// TwinCAT 3 PLC project TwinCAT_OpenFramework_Timers
// Title: TwinCAT Open Framework Timers
// Company: Oleksandr Tiutyk FOP
// Author: Oleksandr Tiutyk
// ProjectVersion: 1.0.13.0
// Description: TwinCAT.OpenFramework object-oriented timer wrapper, works as task
// ProgramVersion: 3.1.4026.28
// libraries:
//   Tc2_Standard, * (Beckhoff Automation GmbH)
//   Tc2_System, * (Beckhoff Automation GmbH)
//   [TwinCAT Open Framework Core], * (Oleksandr Tiutyk FOP)
//   [TwinCAT Open Framework Tasks], * (Oleksandr Tiutyk FOP)
// project tree:
//   Internal/ CurrentNamespace.TcPOU, NamespaceExtractor.TcPOU
//   / ITimer.TcIO, Timer.TcPOU (not stored)
//   Version/ Global_Version.TcGVL
// (motion and I/O tree: see PLC project twincat_openframework_core)
// real-time tasks:
//   TASK PlcTask: cycle T#10ms, priority 20, ADS port 350
//   TASK TestTask: cycle T#10ms, priority 1, ADS port 351
//   TASK RunnerTestTask: cycle T#10ms, priority 2, ADS port 354
//   TASK HowToTask: cycle T#10ms, priority 22, ADS port 353
// variable links:

// ---- Version/Global_Version.TcGVL
{attribute 'TcGenerated'}
{attribute 'no-analysis'}
{attribute 'linkalways'}
// This function has been automatically generated from the project information.
VAR_GLOBAL CONSTANT
	{attribute 'const_non_replaced'}
	stLibVersion_TwinCAT_Open_Framework_Timers : ST_LibVersion := (iMajor := 1, iMinor := 0, iBuild := 13, iRevision := 0, nFlags := 0, sVersion := '1.0.13.0');
END_VAR

// ---- ITimer.TcIO
(*!
<summary>Exposes a task-driven timer's interval, observations and restart operation.</summary>
<description>
Drive the timer through the inherited task lifecycle. Reading observations does not advance time; the
implementation updates them while executing. Timer-specific TON behavior is documented by Timer.
</description>
*)
INTERFACE ITimer EXTENDS TOF_Tasks.ITask

{attribute 'monitoring' := 'call'}
(*!
<summary>Reports the timer's latest elapsed observation.</summary>
<description>
Reading does not update or consume the observation. For Timer this is TON.Q, retained after normal completion
until Reset or restart; it is not independently a successful task-completion result.
</description>
*)
PROPERTY Elapsed : BOOL
GET
END_GET
END_PROPERTY

{attribute 'monitoring' := 'call'}
(*!
<summary>Returns the latest elapsed-time observation without advancing the timer.</summary>
<description>
For Timer this is TON.ET from the most recent TON evaluation, not a live clock read. Reset clears the
observation.
</description>
*)
PROPERTY ElapsedTime : TIME
GET
END_GET
END_PROPERTY

{attribute 'monitoring' := 'call'}
(*!
<summary>Gets or sets the configured timer interval.</summary>
<description>
For Timer, assignment changes TON.PT without a reset, start or immediate observation update. Use
SetIntervalAndRestart to apply an interval and begin timing it from zero.
</description>
*)
PROPERTY Interval : TIME
GET
END_GET
SET
END_SET
END_PROPERTY

(*!
<summary>Prepare a restart, then set the interval and start timing immediately.</summary>
<description>
The method assigns the new interval only after stopping and Reset succeed. A refused preparation returns
FALSE without that assignment; partial effects of descendant callbacks are not rolled back. If Start fails
after preparation, the new interval remains configured. No deferred restart is scheduled. Call outside task
callbacks.
</description>
<param name="interval">Preset for the new run, including zero for completion on its first Execute.</param>
*)

METHOD SetIntervalAndRestart : BOOL
VAR_INPUT
	interval : TIME;
END_VAR
END_METHOD

(*!
<summary>Reports completion in the Execute that observes the timer elapsed.</summary>
<description>
For the ordinary Timer, includes a zero interval and adds no stopping cycle. Read after Execute. The pulse is
cleared by the next Execute, Reset or successful restart; reading does not consume it.
</description>
*)

{attribute 'monitoring' := 'call'}

PROPERTY Triggered : BOOL
GET
END_GET
END_PROPERTY

END_INTERFACE

// ---- Internal/CurrentNamespace.TcPOU
(*
SPDX-FileCopyrightText: © 2026 Oleksandr Tiutyk <trofimich@gmail.com>
SPDX-License-Identifier: MIT
License: https://opensource.org/license/mit
*)

(*!
<summary>Provides this library's namespace text to object metadata getters.</summary>
<description>
Owns the namespace extractor for the program instance's lifetime; no cyclic execution is required.
</description>
*)

{attribute 'no_explicit_call' := 'do not call this POU directly'}
PROGRAM INTERNAL CurrentNamespace
VAR
	{attribute 'hide'} 
	_NamespaceExtractor : NamespaceExtractor;
END_VAR

{attribute 'monitoring' := 'call'}
(*!
<summary>Returns a borrowed reference to the stored namespace text.</summary>
<description>
The reference belongs to this program instance and remains valid while it exists. Callers must treat the text
as read-only; reading does not copy or allocate storage.
</description>
*)
PROPERTY Name : REFERENCE TO STRING
GET
Name REF= _NamespaceExtractor.CurrentNamespace;
END_GET
END_PROPERTY

END_PROGRAM

// ---- Internal/NamespaceExtractor.TcPOU
(*
SPDX-FileCopyrightText: © 2026 Oleksandr Tiutyk <trofimich@gmail.com>
SPDX-License-Identifier: MIT
License: https://opensource.org/license/mit
*)

(*!
<summary>Holds namespace text initialized through the init_namespace attribute.</summary>
<description>
The compiler supplies the initial text; this block performs no runtime extraction or allocation. The owning
CurrentNamespace program exposes the stored text as borrowed metadata.
</description>
*)

FUNCTION_BLOCK INTERNAL NamespaceExtractor
VAR_OUTPUT
	//! <summary>Compiler-initialized namespace storage; consumers must not modify it.</summary>
	{attribute 'init_namespace'} 
	CurrentNamespace : STRING;	
END_VAR

END_FUNCTION_BLOCK
